FUNCTION_BLOCK InputParameter
VAR_INPUT
  interfaceType : InterfaceTypeEnum;
  synchronizationType : SynchronizationTypeEnum;
  discretizationType : DiscretizationTypeEnum;
  
  current_position, current_velocity, current_acceleration : ARRAY[0..ParameterList.MaxDoFs] OF LREAL;
  target_position, target_velocity, target_acceleration : ARRAY[0..ParameterList.MaxDoFs] OF LREAL;
  max_velocity, max_acceleration, max_jerk : ARRAY[0..ParameterList.MaxDoFs] OF LREAL;
  min_velocity, min_acceleration : ARRAY[0..ParameterList.MaxDoFs] OF LREAL;
  
  enabled : ARRAY[0..ParameterList.MaxDoFs] OF BOOL;  
  minDuration : LREAL;
END_VAR
VAR
  dofs_ : INT;
END_VAR

METHOD FB_init : BOOL
VAR_INPUT
	bInitRetains : BOOL; // if TRUE, the retain variables are initialized (warm start / cold start)
	bInCopyCode : BOOL;  // if TRUE, the instance afterwards gets moved into the copy code (online change)
  dofs : INT;
END_VAR
VAR
  i : INT;
END_VAR
dofs_ := dofs;
FOR i:=0 TO ParameterList.MaxDoFs
DO
  enabled[i] := i < dofs;
END_FOR
END_METHOD

END_FUNCTION_BLOCK

(* stored: Version 1.1.0.1, ProductVersion 3.1.4024.9
   POU InputParameter: Id {0a019405-401a-4d00-873d-f46c1ea6dfef}, SpecialFunc None
   Method FB_init: Id {60bc6480-6df7-4a21-b7d6-793f6995b206} *)
